// TIA Portal V16 export
// export: Created 2022-11-17T11:55:29.721644Z, ExportSetting WithDefaults, DisplayName Totally Integrated Automation Portal, DisplayVersion V16 Update 6, DisplayName TIA Portal Version Control Interface, DisplayVersion V16 Update 2, DisplayName TIA Portal Openness, DisplayVersion V16 Update 6, DisplayName SINAMICS Startdrive Advanced, DisplayVersion V16 Update 5, DisplayName SINAMICS Startdrive G130, G150, S120, S150, SINAMICS MV, S210, DisplayVersion V16 Update 5, DisplayName SINAMICS Startdrive G110M, G120, G120C, G120D, G120P, G115D, DisplayVersion V16 Update 5, DisplayName STEP 7 Professional, DisplayVersion V16 Update 6, DisplayName STEP 7 Safety, DisplayVersion V16, DisplayName WinCC Advanced, DisplayVersion V16 Update 6
DATA_BLOCK "DB50_Config"   // DB50
{ S7_Optimized_Access := 'FALSE' }
VERSION : 0.1
// stored: AutoNumber false, IsOnlyStoredInLoadMemory false, IsWriteProtectedInAS false
   VAR RETAIN
      Sel1_Clamp : Int := 3;
      Sel2_BarrierIn : Int := 2;
      Sel3_Pressure : Int := 1;
      Sel4_Doors : Int := 0;
      Sel5_Carriage : Int := 1;
      Sel6_Selfcenter : Int := 2;
      Sel7_Top : Int := 1;
      Sel8_Rope : Int := 3;
      Sel9_BarrierOut : Int := 2;
      Sel10_Conv : Int := 16;
      Sel_Door : Bool := TRUE;
      Sel_EsaurFilm : Bool := FALSE;
      Sel_spare_bool_1 : Bool := FALSE;
      Sel_spare_bool_2 : Bool := FALSE;
      Sel_spare_bool_3 : Bool := FALSE;
      Sel_spare_bool_4 : Bool := FALSE;
      Sel_spare_bool_5 : Bool := FALSE;
      Sel_spare10 : Byte := 16#00;
      Sel_spare11 : Int := 0;
      Sel_spare12 : Int := 0;
      Sel_spare13 : Int := 0;
      Sel_spare14 : Int := 0;
      Sel_spare15 : Int := 0;
      Sel_spare16 : Int := 0;
      Sel_spare17 : Int := 0;
      Sel_spare18 : Int := 0;
      Sel_spare19 : Int := 0;
      Sel_spare20 : Int := 0;
      Sel_spare21 : Int := 0;
      Sel_spare22 : Int := 0;
      Sel_spare23 : Int := 0;
      Sel_spare24 : Int := 0;
      TimerPageFw : Bool := FALSE;
      TimerPageBkw : Bool := FALSE;
   END_VAR
BEGIN
END_DATA_BLOCK
